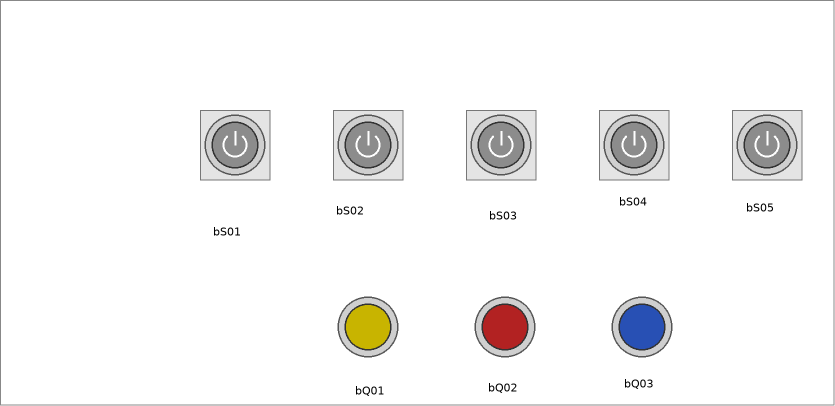
VISUALIZATION Visu  // 835x406
    PowerSwitch (200,110 70x70), variable: MAIN.bS01, behaviour: TOGGLE, style: Switch-PowerSwitch-Gray
    PowerSwitch (333,110 70x70), variable: MAIN.bS02, behaviour: TOGGLE, style: Switch-PowerSwitch-Gray
    PowerSwitch (466,110 70x70), variable: MAIN.bS03, behaviour: TOGGLE, style: Switch-PowerSwitch-Gray
    PowerSwitch (599,110 70x70), variable: MAIN.bS04, behaviour: TOGGLE, style: Switch-PowerSwitch-Gray
    PowerSwitch (732,110 70x70), variable: MAIN.bS05, behaviour: TOGGLE, style: Switch-PowerSwitch-Gray
    Lamp1 (333,292 70x70), variable: MAIN.bQ01, style: Lamp-Lamp1-Yellow
    Lamp1 (470,292 70x70), variable: MAIN.bQ02, style: Lamp-Lamp1-Red
    Lamp1 (607,292 70x70), variable: MAIN.bQ03, style: Lamp-Lamp1-Blue
    Label (152,217 150x30), "bS01"
    Label (275,196 150x30), "bS02"
    Label (564,369 150x30), "bQ03"
    Label (428,373 150x30), "bQ02"
    Label (295,376 150x30), "bQ01"
    Label (428,201 150x30), "bS03"
    Label (558,187 150x30), "bS04"
    Label (685,193 150x30), "bS05"
END_VISUALIZATION

(* stored: Version 1.1.0.1, ProductVersion 3.1.4024.12
   Visu Visu: Id {9db0dd3d-b823-4070-9779-cb85aa3587fe} *)
